TYPE E_ProductFlowState :
(
	none := 0,
	busy,
	done,
	error
);
END_TYPE

(* stored: Version 1.1.0.1, ProductVersion 3.1.0.19
   DUT E_ProductFlowState: Id {f3562ed4-182d-4349-ba9c-8c7c2e45962f} *)
